Staubli VAL3: link_it.pgx

public program link_it(string x_sName)
begin
  // link the point
  // put the base config
end
